{attribute 'linkalways'} 
{attribute 'no_explicit_call' := 'This FB is a CLASS and must be accessed using methods or properties'}
{attribute 'enable_dynamic_creation'}
FUNCTION_BLOCK Node_F_VN_MedianElementElementwise_TcVnVector2_DINT EXTENDS VisionNode
VAR
    ipContainer : _ITcVnContainer;
    aMedian : _TcVnVector2_DINT;
    hrPrev : _HRESULT(S_OK);
    hresult : _HRESULT(S_OK);
END_VAR

METHOD PUBLIC  Clone : I_Node
VAR
	pNode : POINTER TO Node_F_VN_MedianElementElementwise_TcVnVector2_DINT;
END_VAR
pNode := __NEW(Node_F_VN_MedianElementElementwise_TcVnVector2_DINT);
Clone := pNode^;
END_METHOD

METHOD FB_init : BOOL
VAR_INPUT
	bInitRetains : BOOL; // if TRUE, the retain variables are initialized (warm start / cold start)
	bInCopyCode : BOOL;  // if TRUE, the instance afterwards gets moved into the copy code (online change)
END_VAR
AddInput('ipContainer', ipContainer);
AddInput('aMedian', aMedian);
AddInput('hrPrev', hrPrev);
AddOutput('ipContainer', ipContainer);
AddOutput('hresult',hresult);
END_METHOD

METHOD PROTECTED OnExecute : HRESULT
hresult.Value := F_VN_MedianElementElementwise_TcVnVector2_DINT(
    ipContainer := ipContainer.Value,
    aMedian := aMedian.Value,
    hrPrev:= hrPrev.Value);
END_METHOD

METHOD PUBLIC PreExecutionCheck
VAR_INPUT
	Check : I_PreExecutionChecks;
END_VAR
Check.IsTrue(ipContainer.IsValid, 'ipContainer must be a valid container');
END_METHOD

END_FUNCTION_BLOCK

(* stored: Version 1.1.0.1, ProductVersion 3.1.4024.13
   POU Node_F_VN_MedianElementElementwise_TcVnVector2_DINT: Id {807214f0-2713-48fd-9118-91b13e1d9d52}, SpecialFunc None
   Folder Constructor: Id {97b7f373-e2cb-475c-8bef-846679c2e2fc}
   Method Clone: Id {1c596040-5d90-4444-9b07-4909210c5d1b}
   Method FB_init: Id {5d4ce33b-49ec-45ad-9d78-4817c0365511}
   Method OnExecute: Id {9cfd4217-4470-4cd1-8a6d-fed1b26486b8}
   Method PreExecutionCheck: Id {b18ceb8c-a8bb-4ebc-af90-880e8ff18260} *)
